// TIA Portal V21 export
VAR_GLOBAL   // PLC tag table "K_Paratia"
END_VAR
